FUNCTION_BLOCK PUBLIC HRL_NMethod_Auslagern
VAR_INPUT
	NotAusSignal: BOOL;
	LS01_Start: BOOL;
	LS02_Ende: BOOL;
END_VAR
VAR_OUTPUT
	Motor_Auslagern: BOOL;
	Status: BOOL;
END_VAR
VAR
	Transport_Auslagern: Transport_Unidirectional;
	Input_C: BOOL;
	R_TRIG: R_TRIG;
END_VAR

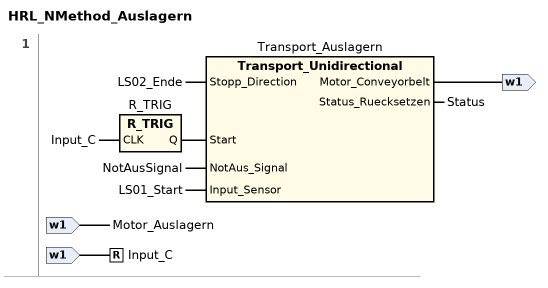
// NETWORK 1
R_TRIG(CLK := Input_C);
Transport_Auslagern(
    Stopp_Direction := LS02_Ende,
    Start := R_TRIG.Q,
    NotAus_Signal := NotAusSignal,
    Input_Sensor := LS01_Start,
    Status_Ruecksetzen => Status); // Transport_Unidirectional
Motor_Auslagern := Transport_Auslagern.Motor_Conveyorbelt;
Input_C R= Transport_Auslagern.Motor_Conveyorbelt;

{attribute 'TcRpcEnable' := '1'}
METHOD METH_Auslagern : BOOL
VAR_INPUT
	MethodCall_C : BOOL;
END_VAR
Input_C := MethodCall_C;
END_METHOD

END_FUNCTION_BLOCK

(* stored: Version 1.1.0.1, ProductVersion 3.1.4024.15
   POU HRL_NMethod_Auslagern: Id {0aaeafec-1005-4ea9-9715-fe32d29acd6c}, SpecialFunc None
   Method METH_Auslagern: Id {5a88dd8a-2d2b-4a3b-b2a3-da836d506e51} *)
